(* IEC 61131-3 sources: AXOpen/src/inspectors/ctrl/src, 5 files *)

(* ---- AxoComprehensiveResult.st ---- *)
NAMESPACE AXOpen.Inspectors

    USING System.Strings;

    ///<summary>
    /// Class for gathering overall result of single or multiple inspections
    /// Only fail results are automatically written to comprehensive result
    /// Application programmer must specify, what is a correct result
    ///</summary>
    {S7.extern=ReadWrite}
    CLASS AxoComprehensiveResult IMPLEMENTS IAxoComprehensiveResult
        VAR PUBLIC

            Result : eOverallResult;
            Failures : STRING;
            ErrorCodes : STRING;

        END_VAR

        ///<summary>
        /// Get the overall result
        ///</summary>
        METHOD PUBLIC GetResult : eOverallResult
            GetResult := Result;
        END_METHOD

        ///<summary>
        /// Get Failures
        /// TODO: not implemented yet
        ///</summary>
        METHOD PUBLIC GetFailures : STRING
            GetFailures := Failures;
        END_METHOD

        ///<summary>
        /// Get error codes
        /// TODO: not implemented yet
        ///</summary>
        METHOD PUBLIC GetErrorCodes : STRING
            GetErrorCodes := ErrorCodes;
        END_METHOD

        ///<summary>
        /// Set overall result
        ///</summary>
        METHOD PUBLIC SetResult
            VAR_INPUT
                inResult : eOverallResult;
            END_VAR
            Result := inResult;
        END_METHOD

        ///<summary>
        /// Set failures
        ///</summary>
        METHOD PUBLIC SetFailures
            VAR_INPUT
                inFailures : STRING;
            END_VAR
            Failures := inFailures;
        END_METHOD

        ///<summary>
        /// Set error codes
        ///</summary>
        METHOD PUBLIC SetErrorCodes
            VAR_INPUT
                inErrorCodes : STRING;
            END_VAR

            ErrorCodes := inErrorCodes;
        END_METHOD

         ///<summary>
        /// Add failure
        ///</summary>
        METHOD PUBLIC AddFailure
            VAR_INPUT
                inFailure : STRING;
            END_VAR

            if (Failures <> '') then
                Failures := Concat(Failures , ';' , inFailure);
            else
                Failures := inFailure;
            end_if;

        END_METHOD

        ///<summary>
        /// Add error code
        ///</summary>
        METHOD PUBLIC AddErrorCode
            VAR_INPUT
                inErrorCode : STRING;
            END_VAR

             if ( ErrorCodes  <> '') then
                ErrorCodes := Concat(ErrorCodes , ';' , inErrorCode);
            else
                ErrorCodes := inErrorCode;
            end_if;
        END_METHOD

    END_CLASS

END_NAMESPACE

(* ---- AxoInspector.st ---- *)
USING AXOpen.Core;
USING System.Strings;

NAMESPACE AXOpen.Inspectors

    ///<summary>
    /// AxoInspector base class with implemented evaluation methods.
    /// Provides methods for checking conditions and invoking inspection tasks.
    ///</summary>
    {S7.extern=ReadWrite}
    CLASS AxoInspector EXTENDS AXOpen.Core.AxoObject IMPLEMENTS IInspector, IOnFail
        VAR PROTECTED
            {#ix-attr:[CompilerOmits("POCO")]} //-"No params" Will skip the emission for all output types
            _inspectorTask: AxoInspectorTask;
            _coordinator: IAxoCoordinator;
            _isOverInspected: BOOL;
            _busy : BOOL;
            _commonData: REF_TO AxoInspectorData;

            _comprehensiveResult      : IAxoComprehensiveResult;
            _comprehensiveResultUpdateCycle    : ULINT; // when was updated comprehensiver result

            _updateOverallResult    : BOOL; // true if is called  UpdateComprehensiveResult()
            _FailureDescription    : STRING; // fill in UpdateComprehensiveResult()
            _ErrorCode             : STRING; // fill in UpdateComprehensiveResult()

        END_VAR

        VAR PUBLIC
            {#ix-attr:[CompilerOmits("POCO")]} //-"No params" Will skip the emission for all output types
            _DL :  AXOpen.Inspectors.AxoInspectorDialog;
        END_VAR

        /// <summary>
        /// Check if the inspection data indicates that the maximum number of retries has been reached.
        /// Returns TRUE if overinspected.
        /// </summary>
        METHOD PUBLIC CheckOverInspection : BOOL
            //check if reference is valid
            IF _inspectorTask.InspectionData() <> NULL THEN
                CheckOverInspection := (_inspectorTask.InspectionData()^.RetryAttemptsCount >= _inspectorTask.InspectionData()^.NumberOfAllowedRetries)
                AND (_inspectorTask.InspectionData()^.NumberOfAllowedRetries <> UINT#0);
            END_IF;
        END_METHOD

        /// <summary>
        /// Calls CheckOverInspection and, if TRUE, invokes the inspection task.
        /// Updates internal flag _isOverInspected.
        /// </summary>
        METHOD PROTECTED IsOverInspected : BOOL
            // Documentation: Evaluate if inspection should be terminated due to excessive retries.
            _isOverInspected := THIS.CheckOverInspection();
            IF(THIS.CheckOverInspection()) THEN
                _inspectorTask.Invoke();
                IF(_inspectorTask.Execute()) THEN
                    _inspectorTask.InspectionData()^.Result := eInspectorResult#Failed;
                    _inspectorTask.DoneWhen(TRUE);
                END_IF;
            END_IF;
            IsOverinspected := THIS.CheckOverInspection();
        END_METHOD

        ///<summary>
        /// Sets the coordinator instance required by the inspector.
        /// </summary>
        METHOD PUBLIC WithCoordinator : IInspector
            VAR_INPUT
                inCoordinator : IAxoCoordinator;
            END_VAR
            // Documentation: Assign the provided coordinator and return the current instance.
            _coordinator := inCoordinator;
            WithCoordinator := THIS;
        END_METHOD

        ///<summary>
        /// Returns this object defined by IOnFail interface.
        /// </summary>
        METHOD PUBLIC OnFail : IOnFail
            // Documentation: If no coordinator is set, the caller is advised to use WithCoordinator.
            OnFail:= THIS;
        END_METHOD

        ///<summary>
        /// Calls the inspector dialog with specified retry and terminate steps.
        /// </summary>
        METHOD PUBLIC Dialog : BOOL
            VAR_INPUT
                inRetryStep: IAxoStep;
                inTerminateStep: IAxoStep;
            END_VAR
            // Documentation: Ensure the coordinator is set before showing the dialog.
            _DL.SetSuspendCyclicExecuteIsNotCalledCheck(TRUE);
            _DL.SetSuspendMultipleExecuteCallCheck(TRUE);
            _DL.Show(REF(THIS), inRetryStep, inTerminateStep);
        END_METHOD

        ///<summary>
        /// If inspection has failed, retries the inspection with the provided step.
        /// </summary>
        METHOD PUBLIC RetryWithStep : BOOL
            VAR_INPUT
                inRetryStep : IAxoStep;
            END_VAR
            // Documentation: Check for coordinator existence. If failed, request the retry step.
            IF(_coordinator = NULL) THEN
                RETURN;
            END_IF;
            IF(THIS.Done()) THEN
                IF(THIS.Result() = eInspectorResult#Failed) THEN
                    IF(inRetryStep <> NULL) THEN
                        _coordinator.RequestStep(inRetryStep);
                        THIS.RestoreInspectorTask();
                    END_IF;
                ELSE
                    _coordinator.MoveNext();
                    THIS.Restore();
                END_IF;
                RetryWithStep:= TRUE;
            END_IF;
        END_METHOD

        METHOD PUBLIC Restore
            _inspectorTask.Restore();

            _comprehensiveResultUpdateCycle := ULINT#0;

            _updateOverallResult := false;
            _FailureDescription :='';
            _ErrorCode :='';
        END_METHOD

        ///<summary>
        /// Continues to the next step when the inspection is completed.
        /// </summary>
        METHOD PUBLIC CarryOn : BOOL
            // Documentation: Verify that the coordinator is set and then move to the next step.
            IF(_coordinator = NULL) THEN
                RETURN;
            END_IF;
            IF(THIS.Done()) THEN

                THIS.UpdateOverallResult();
                _coordinator.MoveNext();
                THIS.Restore();
                CarryOn := TRUE;

            END_IF;
        END_METHOD

        ///<summary>
        /// Terminates the coordination sequence with the provided step when the inspection fails.
        /// </summary>
        METHOD PUBLIC TerminateWithStep : BOOL
            VAR_INPUT
                inTerminateStep : AXOpen.Core.IAxoStep;
            END_VAR
            // Documentation: Terminate by requesting the terminate step or moving on based on inspection result.
            IF(_coordinator = NULL) THEN
                RETURN;
            END_IF;
            IF(THIS.Done()) THEN
                 THIS.UpdateOverallResult();

                IF(THIS.Result() = eInspectorResult#Failed) THEN
                    IF(inTerminateStep <> NULL) THEN
                        _coordinator.RequestStep(inTerminateStep);
                        THIS.RestoreInspectorTask();
                    END_IF;
                ELSE
                    _coordinator.MoveNext();
                    THIS.Restore();
                END_IF;
                TerminateWithStep := TRUE;
            END_IF;
        END_METHOD

        ///<summary>
        /// Updates comprehensive result. The comprehensive result is set to `Failed` when any inspection fails or is inconclusive.
        /// Any bypassed or excluded inspections are not taken into account.
        ///</summary>
        METHOD PUBLIC UpdateComprehensiveResult : IInspector
            VAR_INPUT
                inResult                : IAxoComprehensiveResult;
                inFailureDescription    : STRING;
                inErrorCode             : STRING;
            END_VAR

            _updateOverallResult := true;
            _FailureDescription := inFailureDescription;
            _ErrorCode := inErrorCode;
            _comprehensiveResult := inResult;

            // Documentation: Set overall result to Failed if any inspection fails or is inconclusive.
            UpdateComprehensiveResult := THIS;
            IF(_inspectorTask.InspectionData() = NULL ) THEN
                inResult.SetResult(eOveralLResult#NoAction);
                RETURN;
            END_IF;

        END_METHOD

         ///<summary>
        /// Called only once when the inspector leaves the step.
        /// </summary>
        METHOD INTERNAL UpdateOverallResult

            // must be requested and valid ITF
            if not _updateOverallResult || _comprehensiveResult = NULL ||  _comprehensiveResultUpdateCycle <> ULINT#0 then
                RETURN;
            end_if;

            _comprehensiveResultUpdateCycle := this.GetContext().OpenCycleCount();

            CASE _inspectorTask.InspectionData()^.Result OF

                eInspectorResult#Failed:

                    _comprehensiveResultUpdateCycle := THIS.GetContext().OpenCycleCount();

                    _comprehensiveResult.SetResult(eOverallResult#Failed);
                    _comprehensiveResult.AddFailure(_FailureDescription);
                    _comprehensiveResult.AddErrorCode(_ErrorCode);

                eInspectorResult#Inconclusive:

                    _comprehensiveResultUpdateCycle := THIS.GetContext().OpenCycleCount();

                    _comprehensiveResult.SetResult(eOverallResult#Failed);
                    _comprehensiveResult.AddFailure(_FailureDescription);
                    _comprehensiveResult.AddErrorCode(_ErrorCode);
            ELSE
                ;
            END_CASE;

        END_METHOD

        ///<summary>
        /// Restores the state of the inspector task.
        /// </summary>
        METHOD PUBLIC RestoreInspectorTask : BOOL
            _inspectorTask.Restore();
        END_METHOD

        ///<summary>
        /// Indicates if the inspector task is currently busy.
        /// </summary>
        METHOD PUBLIC Busy : BOOL
            Busy := _inspectorTask.IsBusy();
        END_METHOD

        ///<summary>
        /// Returns the common data associated with this inspector.
        /// </summary>
        METHOD PUBLIC CommonData : REF_TO AXOpen.Inspectors.AxoInspectorData
            CommonData := _commonData;
        END_METHOD

        ///<summary>
        /// Returns the current coordinator.
        /// </summary>
        METHOD PUBLIC Coordinator : IAxoCoordinator
            Coordinator := _coordinator;
        END_METHOD

        ///<summary>
        /// Checks if the inspection task has been completed.
        /// </summary>
        METHOD PUBLIC Done : BOOL
            Done := _inspectorTask.IsDone();
        END_METHOD

        ///<summary>
        /// Returns the result of the inspection.
        /// </summary>
        METHOD PUBLIC Result : eInspectorResult

        VAR
            _inspectorData :  REF_TO AxoInspectorData;
        end_var

        // it can be null
        _inspectorData := _inspectorTask.InspectionData();

        if _inspectorData <> NULL THEN
            Result := _inspectorData^.Result;
        ELSE
            Result := eInspectorResult#NoAction;
        END_IF;

        END_METHOD

        METHOD PRIVATE UpdateDialogInfo
            VAR
                _step : REF_TO AxoStep;
            END_VAR
            IF(_coordinator <> NULL) THEN
                _step ?= _coordinator.GetCurrentStep();
                IF(_step <> NULL) THEN
                    _DL._inspectionDetails := _step^.Descr;
                END_IF;
            END_IF;
        END_METHOD

        /// <summary>
        /// Implements the analog inspection logic.
        /// </summary>
        METHOD PUBLIC Inspect : IInspector
            VAR_INPUT
                inParent : AXOpen.Core.IAxoObject;
                inData : REF_TO AxoAnalogueInspectorData;
                Status : LREAL;
            END_VAR

            VAR
                tmpResult : BOOL;
                _minimum : LREAL;
                _value : LREAL;
                _maximum : LREAL;
                _lastOutValue : LREAL;
                _step : REF_TO AxoStep;
            END_VAR
            VAR CONSTANT
                epsilon : REAL := 10000;
            END_VAR

            _DL._inspectorType := eInspectorType#Analogue;
            _DL._analogInspectorData := inData^;

            // Documentation: Initialize the parent context and the associated inspector task.
            THIS.Run(inParent);
            _inspectorTask.SetSuspendMultipleExecuteCallCheck(TRUE);
            _inspectorTask.SetSuspendCyclicExecuteIsNotCalledCheck(TRUE);
            _inspectorTask.Run(inParent);

            Inspect := THIS;
            _inspectorTask.SetInspectionData(inData);
            IF(THIS.IsOverInspected())THEN
                RETURN;
            END_IF;
            _inspectorTask.Invoke();
            IF (_inspectorTask.Execute()) THEN
                IF (inData^.IsByPassed) THEN
                    inData^.Result    := eInspectorResult#Bypassed;
                    inData^.TimeStamp := THIS.GetContext().GetRtc().NowUTC();
                    _inspectorTask.DoneWhen(TRUE);
                    RETURN;
                END_IF;
                inData^.Result := eInspectorResult#Running;
                _minimum := (inData^.RequiredMin * epsilon);
                _value := (Status * epsilon);
                _maximum := (inData^.RequiredMax * epsilon);
                inData^.DetectedStatus := Status;
                tmpResult := (_minimum <= _value) AND (_maximum >= _value);
                IF(NOT tmpResult) THEN
                    _lastOutValue := Status;
                END_IF;
                _inspectorTask._failTimer.OnDelay(THIS.GetContext(), TRUE, inData^.FailTime);
                _inspectorTask._passTimer.OnDelay(THIS.GetContext(), tmpResult, inData^.PassTime);
                IF(_inspectorTask._passTimer.output OR _inspectorTask._failTimer.output) THEN
                    _inspectorTask.DoneWhen(TRUE);
                    IF (inData^.Result = eInspectorResult#Failed) THEN
                        inData^.DetectedStatus := _lastOutValue;
                        _DL._inspectionDetails := System.Strings.Concat('min:', ToString(inData^.RequiredMin), ' max: ', ToString(inData^.RequiredMax));
                        _DL._inspectionDetails := System.Strings.Concat(_DL._inspectionDetails, ' but was: ', ToString(inData^.DetectedStatus));
                    END_IF;
                    THIS.OnDone();
                    THIS.UpdateDialogInfo();
                END_IF;
            END_IF;
        END_METHOD

        /// <summary>
        /// Implements the string-based inspection logic.
        /// </summary>
        METHOD PUBLIC Inspect : IInspector
            VAR_INPUT
                inParent : AXOpen.Core.IAxoObject;
                inData : REF_TO AxoDataInspectorData;
                Status : STRING;
            END_VAR

            VAR
                tmpResult : BOOL;
                charIndex: DINT;
                charRequired : CHAR;
                charAcquired : CHAR;
                _lastOutValue : STRING;
            END_VAR

            VAR CONSTANT
                epsilon : REAL := 1;
            END_VAR

            _DL._inspectorType := eInspectorType#Data;
            _DL._dataInspectorData := inData^;

            THIS.Run(inParent);
            _inspectorTask.SetSuspendMultipleExecuteCallCheck(TRUE);
            _inspectorTask.SetSuspendCyclicExecuteIsNotCalledCheck(TRUE);
            _inspectorTask.Run(inParent);

            Inspect := THIS;
            _inspectorTask.SetInspectionData(inData);
            IF(THIS.IsOverInspected())THEN
                RETURN;
            END_IF;
            _inspectorTask.Invoke();
            IF (_inspectorTask.Execute()) THEN
                IF (inData^.IsByPassed) THEN
                    inData^.Result    := eInspectorResult#Bypassed;
                    inData^.TimeStamp := THIS.GetContext().GetRtc().NowUTC();
                    _inspectorTask.DoneWhen(TRUE);
                    RETURN;
                END_IF;

                inData^.Result := eInspectorResult#Running;
                inData^.DetectedStatus := Status;
                IF(inData^.StarNotationEnabled) THEN
                    tmpResult := TRUE;
                    // iterate throug the string
                    FOR charIndex := DINT#1 TO LengthOf(inData^.RequiredStatus) DO
                        charRequired := inData^.RequiredStatus[charIndex];
                        IF(LengthOf(inData^.DetectedStatus) >= charIndex) THEN
                            charAcquired :=  inData^.DetectedStatus[charIndex];
                        END_IF;
                        IF(charRequired <> '*' AND charRequired <> '#') THEN
                            tmpResult := charRequired = charAcquired;
                        ELSIF(charRequired = '#') THEN
                            tmpResult := THIS.IsCharNumber(charAcquired);
                        END_IF;
                        IF(NOT tmpResult) THEN
                            EXIT;
                        END_IF;
                    END_FOR;
                ELSE
                    //TODO what about spaces at the beginning and the end?
                    tmpResult := inData^.DetectedStatus = inData^.RequiredStatus;
                END_IF;

                IF(NOT tmpResult) THEN
                    _lastOutValue := Status;
                END_IF;

                _inspectorTask._failTimer.OnDelay(THIS.GetContext(), TRUE, inData^.FailTime);
                _inspectorTask._passTimer.OnDelay(THIS.GetContext(), tmpResult, inData^.PassTime);

                IF(_inspectorTask._passTimer.output OR _inspectorTask._failTimer.output) THEN
                    _inspectorTask.DoneWhen(TRUE);
                    IF (inData^.Result = eInspectorResult#Failed) THEN
                        inData^.DetectedStatus := _lastOutValue;
                        _DL._inspectionDetails := System.Strings.Concat('Req: ', inData^.RequiredStatus);
                        _DL._inspectionDetails := System.Strings.Concat(_DL._inspectionDetails, 'Actual: ', inData^.RequiredStatus);
                    END_IF;
                    THIS.OnDone();
                    THIS.UpdateDialogInfo();
                END_IF;
            END_IF;
        END_METHOD

        /// <summary>
        /// Implements the digital inspection logic.
        /// </summary>
        METHOD PUBLIC Inspect : IInspector
            VAR_INPUT
                inParent : AXOpen.Core.IAxoObject;
                inData : REF_TO AxoDigitalInspectorData;
                Status : BOOL;
            END_VAR

            _DL._inspectorType := eInspectorType#Digital;
            _DL._digitalInspectorData := inData^;

            THIS.Run(inParent);
            _inspectorTask.SetSuspendMultipleExecuteCallCheck(TRUE);
            _inspectorTask.SetSuspendCyclicExecuteIsNotCalledCheck(TRUE);
            _inspectorTask.Run(inParent);

            Inspect := THIS;
            _inspectorTask.SetInspectionData(inData);

            IF(THIS.IsOverInspected()) THEN
                RETURN;
            END_IF;

            _inspectorTask.Invoke();

            IF (_inspectorTask.Execute()) THEN
                IF (inData^.IsByPassed) THEN

                    inData^.Result    := eInspectorResult#Bypassed;

                    inData^.TimeStamp := THIS.GetContext().GetRtc().NowUTC();

                    _inspectorTask.DoneWhen(TRUE);
                    RETURN;
                END_IF;
                inData^.Result := eInspectorResult#Running;
                _inspectorTask._failTimer.OnDelay(THIS.GetContext(), TRUE, inData^.FailTime);
                _inspectorTask._passTimer.OnDelay(THIS.GetContext(), Status = inData^.RequiredStatus, inData^.PassTime);
                inData^.DetectedStatus := Status;
                IF(_inspectorTask._failTimer.output OR _inspectorTask._passTimer.output) THEN
                    _inspectorTask.DoneWhen(TRUE);
                    IF (inData^.Result = eInspectorResult#Failed) THEN
                        inData^.DetectedStatus := NOT inData^.RequiredStatus;
                        _DL._inspectionDetails := System.Strings.Concat('Req: ', ToString(inData^.RequiredStatus));
                        _DL._inspectionDetails := System.Strings.Concat(_DL._inspectionDetails, 'Actual: ', ToString(inData^.RequiredStatus));
                    END_IF;
                    THIS.OnDone();
                    THIS.UpdateDialogInfo();
                END_IF;
            END_IF;
        END_METHOD

        ///<summary>
        /// Called when an inspection is completed.
        /// </summary>
        METHOD OnDone
            ;
        END_METHOD

        ///<summary>
        /// Determines if the provided character is numeric.
        /// </summary>
        METHOD IsCharNumber : BOOL

            VAR_INPUT
                inCharacter: CHAR;
            END_VAR
            IF (inCharacter = '0'
                OR  inCharacter = '1'
                OR  inCharacter = '2'
                OR  inCharacter = '3'
                OR  inCharacter = '4'
                OR  inCharacter = '5'
                OR  inCharacter = '6'
                OR  inCharacter = '7'
                OR  inCharacter = '8'
                OR  inCharacter = '9')
                THEN
                    IsCharNumber := TRUE;
                    RETURN;
                END_IF;
            IsCharNumber := FALSE;
        END_METHOD
    END_CLASS

END_NAMESPACE

(* ---- AxoInspectorData.st ---- *)
NAMESPACE AXOpen.Inspectors

    ///<summary>
    /// Data subjected to each inspector instance.
    ///</summary>
    {S7.extern=ReadWrite}
    CLASS AxoInspectorData

        VAR PUBLIC
        //<CommonInspectorDataDeclaration>
        //timestamp of inspection
        {#ix-set:AttributeName = "<#TimeStamp#>"}
        Timestamp: LDATE_AND_TIME;

        //stabilization time, inspection must be success for this period of time
        {#ix-set:AttributeName = "<#Stab.Time#>"}
        PassTime : TIME;

        //timeout, after which inspection fails
        {#ix-set:AttributeName = "<#Timeout#>"}
        FailTime : TIME;

        //result of inspection
        {#ix-set:AttributeName = "<#Result#>"}
        Result : eInspectorResult;

        //inspection will be performed, however result will be omitted in overall result
        {#ix-set:AttributeName = "<#Excluded#>"}
        IsExcluded: BOOL;

        //inspection will be skipped
        {#ix-set:AttributeName = "<#Bypass#>"}
        IsByPassed : BOOL;

        //maximum number of retries of inspection
        {#ix-set:AttributeName = "<#Re-tries#>"}
        NumberOfAllowedRetries : UINT;

        //actual number of retries
        {#ix-set:AttributeName = "<#Attempts#>"}
        RetryAttemptsCount : UINT;
        //</CommonInspectorDataDeclaration>
        END_VAR

    END_CLASS

END_NAMESPACE

(* ---- AxoInspectorDialog.st ---- *)
USING AXOpen.Core;

NAMESPACE AXOpen.Inspectors

    ///<summary>
    /// AxoInspector base class with implemented evaluation methods
    /// Evaluation methods need IAxoCoordinator instance
    ///</summary>
    {S7.extern=ReadWrite}
    CLASS AxoInspectorDialog EXTENDS AXOpen.Core.AxoDialogBase

        VAR PUBLIC
            _isOverInspected : BOOL;
            _dialogueRetry : BOOL;
            _dialogueTerminate : BOOL;
            _dialogueOverride : BOOL;
            _inspectorIndentity : ULINT; //try display inspector inside dialog.
            _inspectionDetails : STRING;
        END_VAR

        VAR PRIVATE
            _lastCall : ULINT;
            _createPlcCycleSpace : BOOL;
        END_VAR

        VAR
            _isActive : BOOL;
            //_dialogIsClosed : BOOL;
            _isAnswerProvided : BOOL;
        END_VAR

        ///<summary>
        /// Method for showing inspector dialog and handling interaction
        ///</summary>
        METHOD PUBLIC Show
            VAR_INPUT
                _parentInspectorRef : REF_TO AxoInspector;
                inRetryStep : IAxoStep;
                inTerminateStep : IAxoStep;
            END_VAR
            VAR
                callCounter : ULINT;
            END_VAR

            IF(_parentInspectorRef = NULL) THEN
                RETURN;
            END_IF;

            THIS.Initialize(_parentInspectorRef^);

            IF _createPlcCycleSpace THEN // create cycle space AFTER RESPONSE
                _createPlcCycleSpace := FALSE;
                RETURN;
            END_IF;

            //Restores when not called for 2+ consecutive cycles of the context.
            callCounter := THIS.GetParent().GetContext().OpenCycleCount();

            if callCounter = _lastCall then //is called in the same cycle, suppose that is a new dialog
                RETURN;
            END_IF;

            IF(callCounter > _lastCall + ULINT#1) THEN
                THIS.Restore();
            END_IF;
            _lastCall := callCounter;

            _isOverInspected := _parentInspectorRef^.CheckOverInspection();

            IF(_parentInspectorRef^.Done()) THEN

                IF(_parentInspectorRef^.Result() = eInspectorResult#Failed) THEN

                    IF (THIS.Status = eAxoTaskState#Ready) THEN
                        _closeSignal := FALSE;
                    END_IF;

                    _inspectorIndentity := _parentInspectorRef^.GetIdentity();
                    THIS.Invoke();
                    SUPER.Execute();

                    IF(_dialogueRetry) THEN
                        _parentInspectorRef^.RetryWithStep(inRetryStep);
                        _isAnswerProvided := TRUE;

                    END_IF;

                    IF(_dialogueTerminate) THEN
                        _parentInspectorRef^.TerminateWithStep(inTerminateStep);
                        _isAnswerProvided := TRUE;

                    END_IF;

                    IF(_dialogueOverride) THEN
                        _parentInspectorRef^.CarryOn();
                        _isAnswerProvided := TRUE;

                    END_IF;

                ELSE

                    IF(_parentInspectorRef^.Coordinator() <> NULL) THEN
                        _parentInspectorRef^.Coordinator().MoveNext();
                    END_IF;

                END_IF;

                // restore this task, when answer is provided and task is done
                IF _isAnswerProvided THEN
                    THIS.Restore();
                    _parentInspectorRef^.RestoreInspectorTask();
                    _isAnswerProvided := FALSE;
                    _createPlcCycleSpace := TRUE;
                END_IF;

            END_IF;
        END_METHOD

        ///<summary>
        /// Restores dialogue
        ///</summary>
        METHOD PUBLIC Restore

            SUPER.Restore();
            _dialogueRetry := FALSE;
            _dialogueTerminate := FALSE;
            _dialogueOverride := FALSE;
        END_METHOD

    END_CLASS

END_NAMESPACE

(* ---- AxoInspectorTask.st ---- *)
USING AXOpen.Core;
USING AXOpen.Inspectors;
USING AXOpen.Core;

NAMESPACE AXOpen.Inspectors

    {S7.extern=ReadWrite}
    CLASS AxoInspectorTask EXTENDS AxoTask
        VAR
            _onDoneFlag: BOOL;
            _inspectionData: REF_TO AxoInspectorData;

        END_VAR

        VAR INTERNAL
            _passTimer : AXOpen.Timers.OnDelayTimer;
            _failTimer : AXOpen.Timers.OnDelayTimer;
        END_VAR

        //getter
        METHOD PUBLIC InspectionData : REF_TO AxoInspectorData
            InspectionData := _inspectionData;
        END_METHOD

        //setter
        METHOD INTERNAL SetInspectionData : REF_TO AxoInspectorData
            VAR_INPUT
                inInspectionData: REF_TO AxoInspectorData;
            END_VAR
            _inspectionData := inInspectionData;
        END_METHOD

        METHOD PUBLIC OnDoneFlag : BOOL
            OnDoneFlag := _onDoneFlag;
        END_METHOD

        ///<summary>
        /// Execute inspection task.
        ///</summary>
        METHOD PUBLIC OVERRIDE Execute : BOOL
            VAR_INPUT
                inParent : IAxoObject;
            END_VAR;

            _onDoneFlag := FALSE;
            Execute := SUPER.Execute(inParent);
        END_METHOD

        ////<summary>
        /// Executes once when inspection starts.
        ///</summary>
        METHOD PROTECTED OVERRIDE OnStart
            SUPER.OnStart();

            // set default value for failtime if no values were provided
            // minimal pass time is not requested due to evaluation in the same plc cycle
            // IF (_inspectionData^.PassTime = T#0S) THEN
            //     _inspectionData^.PassTime := T#50MS;
            // END_IF;

            IF (_inspectionData^.FailTime = T#0S) THEN
                _inspectionData^.FailTime := T#100MS;
            END_IF;

            _inspectionData^.Result := eInspectorResult#NoAction;

            _passTimer.Restore();
            _failTimer.Restore();
        END_METHOD

        METHOD PUBLIC Restore
            SUPER.Restore();
            _onDoneFlag := FALSE;
        END_METHOD

        ////<summary>
        /// When inspection Task is done, evaluate inspection result and write to inspection data.
        ///</summary>
        METHOD PROTECTED OVERRIDE OnDone
            SUPER.OnDone();

            // iterate number of retries
            _inspectionData^.RetryAttemptsCount := _inspectionData^.RetryAttemptsCount + UINT#1;

            // if inspection is set to be bypassed, skip evalution of result
            IF (_inspectionData^.Result = eInspectorResult#Bypassed) THEN
                RETURN;
            END_IF;

            _inspectionData^.TimeStamp := THIS.GetContext().GetRtc().NowUTC();
            _inspectionData^.Result    := eInspectorResult#Failed;

            // if fail timer was not satisfied and pass timer passed, set inspector result to passed
            IF (NOT _failTimer.output AND _passTimer.output) THEN
                _inspectionData^.Result := eInspectorResult#Passed;
            END_IF;

            // if inspector was excluded, set result to excluded
            IF (_inspectionData^.IsExcluded) THEN
                _inspectionData^.Result := eInspectorResult#Excluded;
            END_IF;

            _onDoneFlag := TRUE;
        END_METHOD

    END_CLASS

END_NAMESPACE
